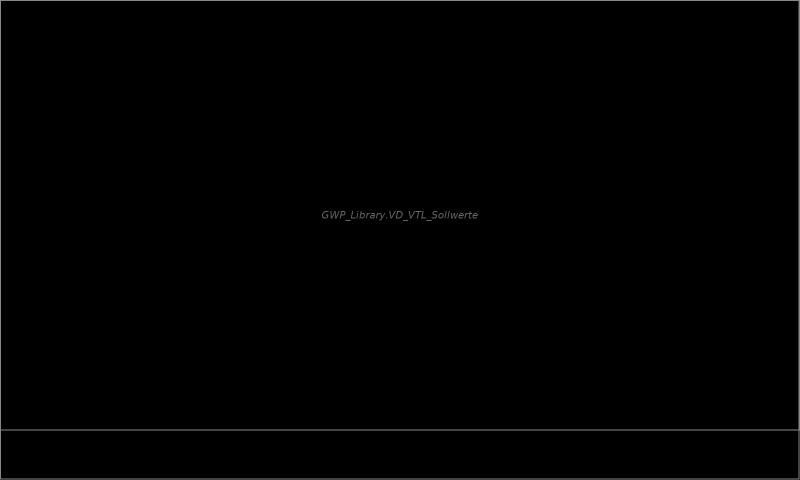
VISUALIZATION VD_VTL_Sollwerte  // 800x480
    Frame (0,0 800x430)
        shows GWP_Library.VD_VTL_Sollwerte(FB_VD := Main.VD_0, FB_Init_1 := Main.Init_0)
END_VISUALIZATION

(* stored: Version 1.1.0.1, ProductVersion 3.1.4022.6
   Visu VD_VTL_Sollwerte: Id {12690779-040b-4f01-b708-2c7ef69e0f06} *)
